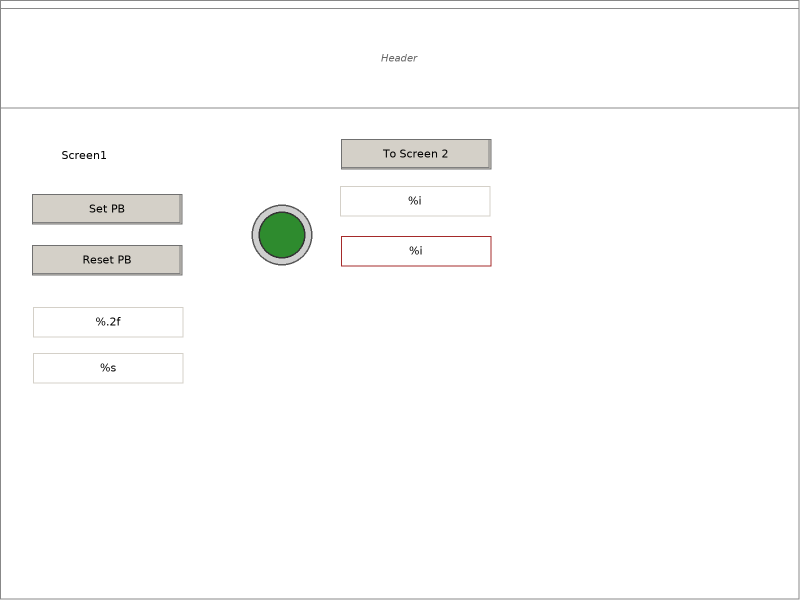
VISUALIZATION Screen1  // 800x600
    Label (32,122 105x67), "Screen1"
    Button (32,194 150x30), "Set PB", colour toggle: GVL.Bool1
        tap GVL.Bool1
    Lamp1 (247,200 70x70), variable: GVL.Bool3, style: Lamp-Lamp1-Green
    Button (32,245 150x30), "Reset PB", colour toggle: GVL.Bool2
        tap GVL.Bool2
    Textfield (340,186 150x30), "%i", text variable: GVL.Number1
        OnMouseDown: write the text variable via VisuDialogs.Numpad
    Textfield (341,236 150x30), "%i", text variable: GVL.Number2
    Textfield (33,307 150x30), "%.2f", text variable: GVL.Real1
    Textfield (33,353 150x30), "%s", text variable: GVL.String1
    Button (341,139 150x30), "To Screen 2"
        OnMouseDown: change screen: Screen2
    Frame (-1,8 800x100)
        shows Header()
END_VISUALIZATION

(* stored: Version 1.1.0.1, ProductVersion 3.1.4024.12
   Visu Screen1: Id {1634b992-a268-4114-9819-e62befad19a4} *)
